(* IEC 61131-3 sources: CodesysTest/export/Function Blocks/IO/FB_PhysicalDigitalOutput.pou, 4 files *)

(* ---- FB_PhysicalDigitalOutput.pou.st ---- *)
(*#-#-#-#-#-#-#-#-#-#---Declaration---#-#-#-#-#-#-#-#-#-#-#-#-#*)

FUNCTION_BLOCK FB_PhysicalDigitalOutput EXTENDS FB_BaseObject IMPLEMENTS ILoggable, ISimulateable
VAR_INPUT
	refOutput : REFERENCE TO BOOL; //  Reference to physical output

END_VAR
VAR_OUTPUT
	Q : BOOL;		// Logical inidcation of output
END_VAR
VAR
	outputONS : FB_ONS;
	_simulate : BOOL;	// Simulate output - do not trigger actual physical output
END_VAR
VAR_IN_OUT

END_VAR
(*#-#-#-#-#-#-#-#-#-#---Implementation---#-#-#-#-#-#-#-#-#-#-#-#-#*)

(* ---- Execute.m.st ---- *)
(*#-#-#-#-#-#-#-#-#-#---Declaration---#-#-#-#-#-#-#-#-#-#-#-#-#*)

METHOD Execute
VAR_INPUT
END_VAR
(*#-#-#-#-#-#-#-#-#-#---Implementation---#-#-#-#-#-#-#-#-#-#-#-#-#*)

outputONS(CLK := Q);

IF __ISVALIDREF(refoutput) THEN
	IF _simulate THEN
		refOutput := FALSE;
	ELSE
		refOutput := Q;
	END_IF
END_IF

IF outputONS.OSR THEN
    _logger.AddLogItem(CONCAT(_prefix, 'On'));
END_IF

IF outputONS.OSF THEN
    _logger.AddLogItem(CONCAT(_prefix, 'Off'));
END_IF

(* ---- TurnOff.m.st ---- *)
(*#-#-#-#-#-#-#-#-#-#---Declaration---#-#-#-#-#-#-#-#-#-#-#-#-#*)

METHOD TurnOff
VAR_INPUT
END_VAR
(*#-#-#-#-#-#-#-#-#-#---Implementation---#-#-#-#-#-#-#-#-#-#-#-#-#*)

Q := FALSE;
Execute();

(* ---- TurnOn.m.st ---- *)
(*#-#-#-#-#-#-#-#-#-#---Declaration---#-#-#-#-#-#-#-#-#-#-#-#-#*)

METHOD TurnOn
VAR_INPUT
END_VAR
(*#-#-#-#-#-#-#-#-#-#---Implementation---#-#-#-#-#-#-#-#-#-#-#-#-#*)

Q := TRUE;
Execute();
